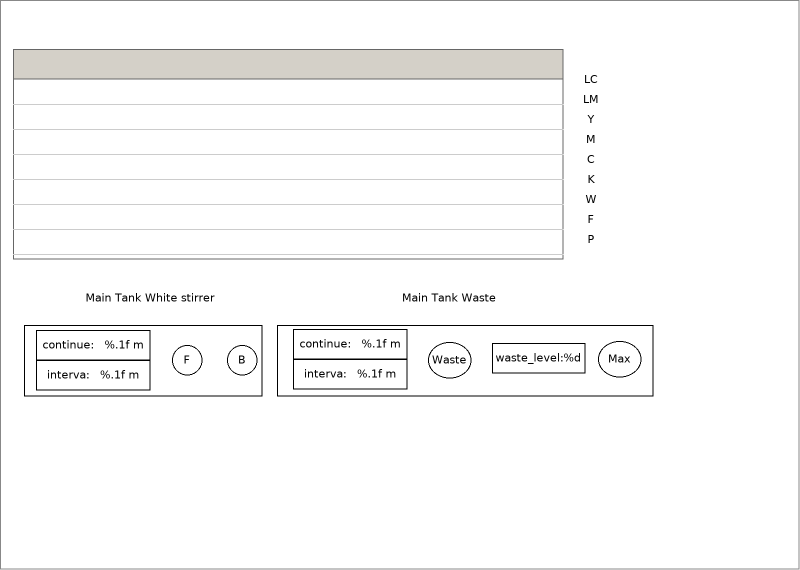
VISUALIZATION VIS_ISS  // 800x570
    RoundedRectangle (277,325 376x71)
    RoundedRectangle (24,325 238x71)
    Table (13,49 550x210), data array: GVL_API.stISS
        p3854506369: GVL_API.stISS[INDEX].error_code
        p1892666644: GVL_API.stISS[INDEX].state
        p338671338: GVL_API.stISS[INDEX].mainTankLevel
        p2170511999: GVL_API.stISS[INDEX].Init_Done
        p3723444502: GVL_API.stISS[INDEX].Error
        p1218418051: GVL_API.stISS[INDEX].Initialize
        p746581629: GVL_API.stISS[INDEX].Setoff
        p3104783080: GVL_API.stISS[INDEX].sensor_blink
        Columns.Column.[5].Template: toggle GVL_API.stISS[INDEX].Initialize
        Columns.Column.[6].Template: toggle GVL_API.stISS[INDEX].Setoff
    Rectangle (36,330 114x30), "continue: %.1f m", text variable: HMI_SetStirrer_continueTime
        OnMouseDown: write HMI_SetStirrer_continueTime via Default, min 0.01
    Rectangle (36,360 114x30), "interva: %.1f m", text variable: HMI_SetStirrer_intervalTime
        OnMouseDown: write HMI_SetStirrer_intervalTime via Default, min 0.5
    Ellipse (172,345 30x30), "F", colour toggle: stOutput.bqStirrerWorkingF
    Ellipse (227,345 30x30), "B", colour toggle: stOutput.bqStirrerWorkingB
    Ellipse (428,342 43x36), "Waste", colour toggle: stOutput.bqWastePump
    Rectangle (293,329 114x30), "continue: %.1f m", text variable: HMI_SetWaste_continueTime
        OnMouseDown: write HMI_SetWaste_continueTime via Default
    Rectangle (293,359 114x30), "interva: %.1f m", text variable: HMI_SetWaste_intervalTime
        OnMouseDown: write HMI_SetWaste_intervalTime via Default, min 0.1
    Rectangle (492,343 93x30), "waste_level:%d", text variable: GVL.MainTankLevel[10]
    Ellipse (598,341 43x36), "Max", colour toggle: GVL_API.stMU.waste_maximum_level
    Label (567,72 48x15), "LC"
    Label (567,92 48x15), "LM"
    Label (567,112 48x15), "Y"
    Label (567,132 48x15), "M"
    Label (567,152 48x15), "C"
    Label (567,192 48x15), "W"
    Label (567,232 48x15), "P"
    Label (567,172 48x15), "K"
    Label (567,212 48x15), "F"
    Label (68,283 164x30), "Main Tank White stirrer"
    Label (367,283 164x30), "Main Tank Waste"
END_VISUALIZATION

(* stored: Version 1.1.0.1, ProductVersion 3.1.4024.11
   Visu VIS_ISS: Id {ac6c71d9-438c-463a-9e81-b59f23470fc4} *)
